FUNCTION_BLOCK GEN_SIN (* this signal generator generates a sine wave output *)
  (* Standard: 61499-1; Description: version 1.6	11. mar. 2009 programmer 	oscat tested BY	oscat this signal generator generates a sine wave output. The sine wave signal is defined by period time (PT), amplitude (AM), offset (OS) and a specific delay for the output signal (DL). The Output waveform will have its max peak at AM/2 + OS and its minimum peak at -AM/2 + OS. The delay input can delay a signal up to PT, this can be useful to synchronize different generators and generate interleaving signals. A Cos wave can be generated accordingly. in addition to a analog output Out there is a second boolean output Q with the corresponding binary signal. *)
  (* Version 1.0, 2025-12-21, franz *)
  PACKAGE OSCAT::Basic::POUs::Engineering::signal_generators;
  IMPORT OSCAT::Basic::Globals::Constants::MATH;
  IMPORT OSCAT::Basic::POUs::Mathematical::MODR;
  IMPORT OSCAT::Basic::POUs::Mathematical::SIGN_R;
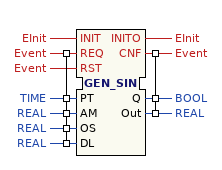
  EVENT_INPUT
    INIT : EInit; (* Init Request *)
    REQ WITH PT, AM, OS, DL; (* Normal Execution Request *)
    RST; (* Reset *)
  END_EVENT
  EVENT_OUTPUT
    INITO : EInit; (* Init Confirmation *)
    CNF WITH Q, Out; (* Execution Confirmation *)
  END_EVENT
  VAR_INPUT
    PT : TIME; (* Period Time *)
    AM : REAL := 1.0; (* Amplitude *)
    OS : REAL; (* Offset *)
    DL : REAL; (* Delay *)
  END_VAR
  VAR_OUTPUT
    Q : BOOL; (* Binary Output *)
    Out : REAL; (* Analog Output *)
  END_VAR
  VAR
    tx : TIME;
    last : TIME;
    init : BOOL;
    temp : REAL;
    DL_M : REAL;
  END_VAR
  EC_STATES
    INIT : INIT -> INITO;
    REQ : REQ -> CNF;
    RST : RST -> CNF;
  END_STATES
  ALGORITHM INIT IN ST:
init := FALSE;
  END_ALGORITHM
  ALGORITHM RST IN ST:
init := TRUE;
last := tx;
tx := T#0s;
  END_ALGORITHM
  ALGORITHM REQ IN ST:
ALGORITHM REQ
(* read system time and prepare input data *)
tx := NOW_MONOTONIC() - last;
DL_M := MODR(DL, 1.0);
IF DL_M < 0.0 THEN
	DL_M := 1.0 - DL_M;
END_IF;

(* init section *)
IF NOT init THEN
	this.RST();
END_IF;

(* add last if one cycle is finished *)
IF tx >= PT THEN
	last := last + PT;
	tx := tx - PT;
END_IF;

(* generate sine wave *)
IF PT > T#0s THEN
	temp := SIN(MATH.PI2 * UDINT_TO_REAL(TIME_IN_MS_TO_UDINT(tx + (PT * DL))) / UDINT_TO_REAL(TIME_IN_MS_TO_UDINT(PT)));
END_IF;
Out := AM * 0.5 * temp + OS;

(* boolean output Q *)
Q := NOT SIGN_R(temp);
END_ALGORITHM

(* revision history hm	22. jan 2007	rev 1.0 original version
 * *
 * hm	17 sep 2007	rev 1.1 replaced time() with t_plc_ms for compatibilitx reasons
 * *
 * hm	27. nov 2007	rev 1.2 avoid divide by 0 when pt = 0
 * *
 * hm	6. jan 2008		rev 1.3 improved performance
 * *
 * hm	16. mar. 2008	rev 1.4 added type conversion to avoid warnings under codesys 3.0
 * *
 * hm	18. oct. 2008	rev 1.5 using math constants
 * *
 * hm	11. mar. 2009	rev 1.6 changed real constants to use dot syntax *)
  END_ALGORITHM
END_FUNCTION_BLOCK
